// TIA Portal V16 export
// export: Created 2022-01-12T14:34:29.0029135Z, ExportSetting WithDefaults, DisplayName Totally Integrated Automation Portal, DisplayVersion V16 Update 4, DisplayName TIA Portal Version Control Interface, DisplayVersion V16 Update 2, DisplayName TIA Portal Openness, DisplayVersion V16 Update 4, DisplayName STEP 7 Professional, DisplayVersion V16 Update 4, DisplayName STEP 7 Safety, DisplayVersion V16, DisplayName WinCC Professional, DisplayVersion V16 Update 4
TYPE "typSygnałObjectToCip"
// stored: IsFailsafeCompliant false
   STRUCT
      iLifeWord : UInt;   // lifeword:=lifeword+1 every 100ms
      iNrOfReadyObjectToCip : UInt;   // identification of ready object to Cip
      bReadyToCip : Bool;   // object is ready to Cip
      bTankisNotEmpty : Bool;   // show low-level sensor if tank is draining
      bReqPause : Bool;   // object request pause of Cip process
      bError : Bool;   // object send Error
   END_STRUCT;
END_TYPE
